PROGRAM MessageProvider
VAR
	Message : ARRAY[0..10] OF STRING;
	FinalMessage : STRING[1000];
	i: INT;
END_VAR



IF RecipeTags.Recipe.Blocks[RecipeControl.nCurrentBlock].Properties.bBlockStarted AND RecipeTags.Recipe.Blocks[RecipeControl.nCurrentBlock].Name='Transfer' THEN
	Message[0] := concat(RecipeTags.Recipe.Blocks[RecipeControl.nCurrentBlock].Name,' - ');
	Message[1] := concat(Message[0], RecipeTags.Recipe.Blocks[RecipeControl.nCurrentBlock].Properties.sSource );
	Message[2] := concat(Message[1],' to ' );
	Message[3] := concat(Message[2], RecipeTags.Recipe.Blocks[RecipeControl.nCurrentBlock].Properties.sDestination);
	Message[4] := concat(Message[3], ' Started At ');
	Message[5] := concat(Message[4], RecipeTags.StaredTimeForRecipeBanner);
	RecipeTags.RecipeMessage := Message[5];
END_IF


IF RecipeTags.Recipe.Blocks[RecipeControl.nCurrentBlock].Properties.bBlockStarted AND RecipeTags.Recipe.Blocks[RecipeControl.nCurrentBlock].Name='Stirrer' THEN
	Message[0] := concat(RecipeTags.Recipe.Blocks[RecipeControl.nCurrentBlock].Name,' - ');
	Message[1] := concat(Message[0], RecipeTags.Recipe.Blocks[RecipeControl.nCurrentBlock].Properties.sSource );
	Message[2] := concat(Message[1], ' Started At ');
	Message[3] := concat(Message[2], RecipeTags.StaredTimeForRecipeBanner);
	RecipeTags.RecipeMessage := Message[3];
END_IF

IF RecipeTags.Recipe.Blocks[RecipeControl.nCurrentBlock].Properties.bBlockStarted AND RecipeTags.Recipe.Blocks[RecipeControl.nCurrentBlock].Name='Drain' THEN
	Message[0] := concat(RecipeTags.Recipe.Blocks[RecipeControl.nCurrentBlock].Name,' - ');
	Message[1] := concat(Message[0], RecipeTags.Recipe.Blocks[RecipeControl.nCurrentBlock].Properties.sSource );
	Message[2] := concat(Message[1], ' Started At ');
	Message[3] := concat(Message[2], RecipeTags.StaredTimeForRecipeBanner);
	RecipeTags.RecipeMessage := Message[3];
END_IF


IF RecipeTags.Recipe.Blocks[RecipeControl.nCurrentBlock].Properties.bBlockStarted AND RecipeTags.Recipe.Blocks[RecipeControl.nCurrentBlock].Name='N2Purge' THEN
	Message[0] := concat(RecipeTags.Recipe.Blocks[RecipeControl.nCurrentBlock].Name,' - ');
	Message[1] := concat(Message[0], RecipeTags.Recipe.Blocks[RecipeControl.nCurrentBlock].Properties.sSource );
	Message[2] := concat(Message[1], ' Started At ');
	Message[3] := concat(Message[2], RecipeTags.StaredTimeForRecipeBanner);
	RecipeTags.RecipeMessage := Message[3];
END_IF


IF RecipeTags.Recipe.Blocks[RecipeControl.nCurrentBlock].Properties.bBlockStarted AND RecipeTags.Recipe.Blocks[RecipeControl.nCurrentBlock].Name='Wait' THEN
	Message[0] := concat(RecipeTags.Recipe.Blocks[RecipeControl.nCurrentBlock].Name,' - ');
	Message[1] := concat(Message[0], RecipeTags.Recipe.Blocks[RecipeControl.nCurrentBlock].Properties.sSource );
	Message[2] := concat(Message[1], ' Started At ');
	Message[3] := concat(Message[2], RecipeTags.StaredTimeForRecipeBanner);
	RecipeTags.RecipeMessage := Message[3];
END_IF

IF RecipeTags.Recipe.Blocks[RecipeControl.nCurrentBlock].Properties.bBlockStarted AND RecipeTags.Recipe.Blocks[RecipeControl.nCurrentBlock].Name='Start' THEN
	Message[0] := concat('Recipe Started At ',RecipeTags.StaredTimeForRecipeBanner);
	RecipeTags.RecipeMessage := Message[0];
END_IF


IF RecipeTags.Recipe.Blocks[RecipeControl.nCurrentBlock].Properties.bBlockStarted AND RecipeTags.Recipe.Blocks[RecipeControl.nCurrentBlock].Name='End' THEN
	Message[0] := concat('Recipe Ended At ',RecipeTags.StaredTimeForRecipeBanner);
	RecipeTags.RecipeMessage := Message[0];
END_IF

IF RecipeTags.Recipe.Blocks[RecipeControl.nCurrentBlock].Name='' THEN
	
	FOR i:=0 TO 10 DO
		Message[i] := ''; 
	END_FOR
	RecipeTags.RecipeMessage := '';
END_IF

END_PROGRAM

(* stored: Version 1.1.0.1, ProductVersion 3.1.4024.5
   POU MessageProvider: Id {1b8a6de6-d39b-459f-baa4-f4f250f34048}, SpecialFunc None *)
